(* CODESYS project plc_chalet_base.library
   Title: CHALET_BaseComponents
   Version: 3.2.4
   Placeholder: CHALET_BaseComponents
   Company: Beckhoff CH

Project tree, tasks and I/O mapping:
  libraries: Tc2_EtherCAT, * (Beckhoff Automation GmbH); Tc2_Standard, 3.3.3.0 (Beckhoff Automation GmbH); Tc2_System, 3.4.25.0 (Beckhoff Automation GmbH); Tc2_Utilities, 3.3.52.0 (Beckhoff Automation GmbH); Tc3_EventLogger, 3.1.30.0 (Beckhoff Automation GmbH); Tc3_Module, 3.3.21.0 (Beckhoff Automation GmbH)
  COMPONENTs/
    CoE-Access/
      internal/
        function block FB_CoE_Base [ST]: cbBufLen, Index, pSrcBuf, SubIndex, Error, FB_init, ReadDone, Update, WriteDone
        interface I_AdsAddr: NetId, Port
      function block FB_CoE_BOOL [ST]: cbBufLen, pSrcBuf, Value
      function block FB_CoE_BYTE [ST]: cbBufLen, pSrcBuf, Value
      function block FB_CoE_Connection [ST]: Mapped, NetId, Port
      function block FB_CoE_UDINT [ST]: cbBufLen, pSrcBuf, Value
      function block FB_CoE_UINT [ST]: cbBufLen, pSrcBuf, Value
    Feedback/
      function block FB_CH_Feedback [ST]: ActiveCommand, Busy, Done, Error, ErrorId, HR, LastCommandAccepted
      interface I_CH_Feedback: ActiveCommand, Busy, Done, Error, ErrorId, HR, LastCommandAccepted
    HR/
      function CheckNotOk [ST]
      function CheckOk [ST]
      function GetMostSignificant [ST]
    List/
      CD_CH_List
      function block FB_CH_List [ST]: FindLUID, FindOID, FindOIDString, ResetIterator, RestoreIterator, AddList, Clear, Duplicate, Initialize, IsEmpty, IsFull, Size, Update, AddObject, FindObject, GetNextObject, GetRandomObject, HasNextObject, RemoveObject
      interface I_CH_LIST: FindLUID, FindOID, FindOIDString, GetNextObject, GetRandomObject, HasNextObject, IsEmpty, IsFull, ResetIterator, RestoreIterator, Size
    Object/
      CD_CH_Object
      function block FB_CH_Object [ST]: FB_init, Initialize, LUID, OID, TaskIndex, Update
      interface I_CH_Object: Initialize, LUID, OID, Update
    global variables GVL_Datatypes
  global variables BaseParameterlist
  00000000-0000-0000-0000-000000000000|LICENSE.md
  LICENSE.md
*)

// COMPONENTs/GVL_Datatypes
{attribute 'qualified_only'}
VAR_GLOBAL CONSTANT
	// SINT
	cMaxSint	: SINT 		:= 127; // Largest SINT number
    cMinSint	: SINT 		:= -128; // Smallest SINT number

	// USINT
	cMaxUsint	: USINT 	:= 255; // Largest USINT number
    cMinUSint	: USINT 	:= 0; // Smallest USINT number

	// INT
	cMaxInt		: INT 		:= 32_767; // Largest INT number
    cMinInt		: INT 		:= -32_768; // Smallest INT number

	// UINT
	cMaxUint	: UINT 		:= 65_535; // Largest UINT number
    cMinUnit	: UINT 		:= 0; // Smallest UINT number

	// DINT
	cMaxDint	: DINT 		:= 2_147_483_647; // Largest DINT number
    cMinDint	: DINT 		:= -2_147_483_648; // Smallest DINT number

	// UDINT
	cMaxUdint	: UDINT 	:= 4_294_967_295; // Largest UDINT number
    cMinUdint	: UDINT		:= 0; // Smallest UDINT number

	// LINT
	cMaxLint	: LINT 		:= 9_223_372_036_854_775_807; // Largest LINT number
    cMinBLint	: LINT 		:= -9_223_372_036_854_775_808; // Smallest LINT number

	// ULINT
	cMaxUlint	: ULINT 	:= 18_446_744_073_709_551_615; // Largest ULINT number
    cMinUlint	: ULINT 	:= 0; // Smallest ULINT number

	// BYTE
	cMaxByte	: BYTE 		:= 255; // Largest BYTE number
    cMinByte	: BYTE 		:= 0; // Smallest BYTE number

	// WORD
	cMaxWord	: WORD 		:= 65_535; // Largest WORD number
    cMinWord	: WORD 		:= 0; // Smallest WORD number

	// DWORD
	cMaxDword	: DWORD 	:= 4_294_967_295; // Largest DWORD number
    cMinDword	: DWORD 	:= 0; // Smallest DWORD number

	// LWORD
	cMaxLword	: LWORD 	:= 18_446_744_073_709_551_615; // Largest LWORD number
    cMinLword	: LWORD 	:= 0; // Smallest LWORD number
	
	// REAL
	cMaxReal	: REAL 		:= 3.402823E+38; // Largest REAL number
    cMinReal	: REAL 		:= -3.402823E+38; // Smallest REAL number
	
	// LREAL
    cMaxLreal	: LREAL 	:= 1.7976931348623157E+308; // Largest LREAL number
    cMinLreal	: LREAL 	:= -1.7976931348623157E+308; // Smallest LREAL number
	
    // DATE
    cMaxDate   	: DATE    	:= DATE#2106-2-7; // Maximum DATA
    cMinDate   	: DATE     	:= DATE#1970-1-1; // Minimum DATE
	
	// TIME
	cMaxTime	: TIME  	:= T#49D17H2M47S295MS; // Longest TIME duration
	cMinTime 	: TIME  	:= TO_TIME(0);	// Shortest TIME duration
	
	// LTIME
	cMaxLtime	: LTIME 	:= LTIME#213503D23H34M33S709MS551US615NS; // Longest LTIME duration
	cMinLtime 	: LTIME  	:= TO_LTIME(0); // Shortest LTIME duration
	
    // Date and time
    cMaxDataAndTime  : DATE_AND_TIME  := DATE_AND_TIME#2106-02-07-06:28:15; // Maximum DATA_AND_DATE
    cMinDataAndTime  : DATE_AND_TIME  := DATE_AND_TIME#1970-1-1-0:0:0; // Minimum DATA_AND_DATE

    // Time of day
    cMaxTimeOfDay 	: TIME_OF_DAY    := TIME_OF_DAY#23:59:59.999; // Largest TIME_OF_DAY
    cMinTimeOfDay 	: TIME_OF_DAY    := TIME_OF_DAY#0:0:0; // Smallest TIME_OF_DAY

END_VAR

// BaseParameterlist
{attribute 'qualified_only'}
VAR_GLOBAL CONSTANT
	(*Maximum length of List*)
	MAX_OBJECTS 			: UDINT := 150;
	
	(*Maximum CoE-Read at same time*)
	MAX_COE_READ 			: UDINT := 20;
	
	(*Maximum CoE-Write at same time*)
	MAX_COE_WRITE 			: UDINT := 20;
	
	
END_VAR

// COMPONENTs/CoE-Access/internal/FB_CoE_Base
(* This FB is abstract and is the base class  *)
FUNCTION_BLOCK ABSTRACT FB_CoE_Base EXTENDS FB_CH_Object
VAR
	//Coe Connector
	{attribute 'hide'}
	ipCoeConnection	: I_AdsAddr;
	{attribute 'hide'}
	bErrorInvalideInterface : BOOL;
	
	//Parameter index
	{attribute 'hide'}
    nIndex     : WORD; (* CoE Object Index *)
	{attribute 'hide'}
    nSubIndex  : BYTE; (* Subindex of CoE Object *)

	//Read/write 
	{attribute 'hide'}
	bReadDone : BOOL;
	{attribute 'hide'}
	fbCoeRead : FB_EcCoeSdoRead;
	{attribute 'hide'}
	nSeqRead : UINT;
	{attribute 'hide'}
	bReadError : BOOL;
	
	{attribute 'hide'}
	bWriteDone : BOOL := TRUE;
	{attribute 'hide'}
	fbCoeWrite : FB_EcCoeSdoWrite;
	{attribute 'hide'}
	nSeqWrite : UINT;
	{attribute 'hide'}
	bWriteError : BOOL;
	
	{attribute 'hide'}
	fbDelayOnError : TON := ( PT:= T#10S);
END_VAR
VAR_STAT
	nCtsCoeObject : UDINT;
	nCtsReadActive : UDINT;
	nCtsWriteActive : UDINT;
END_VAR

PROPERTY PROTECTED ABSTRACT cbBufLen : UDINT
GET
END_GET
END_PROPERTY

PROPERTY PRIVATE Index : WORD
GET
END_GET
END_PROPERTY

PROPERTY PROTECTED ABSTRACT pSrcBuf : PVOID
GET
END_GET
END_PROPERTY

PROPERTY PRIVATE SubIndex : BYTE
GET
END_GET
END_PROPERTY

{attribute 'monitoring':='call'}
PROPERTY Error : BOOL
GET
Error := THIS^.bReadError OR THIS^.bWriteError OR THIS^.bErrorInvalideInterface;
END_GET
END_PROPERTY

METHOD FB_init : BOOL
VAR_INPUT
	bInitRetains : BOOL; // if TRUE, the retain variables are initialized (warm start / cold start)
	bInCopyCode : BOOL;  // if TRUE, the instance afterwards gets moved into the copy code (online change)
	
	ipCoeConnection	: I_AdsAddr;
    nIndex     : WORD; 	(* CoE Object Index *)
    nSubIndex  : BYTE; 		(* Subindex of CoE Object *)
END_VAR

VAR_INST
	{attribute 'hide'}
	bFBInitCalledOnce : BOOL; //Do the following code once during start up and not during onlinechange
END_VAR
//Do the following code once during start up and not during onlinechange
IF NOT bFBInitCalledOnce THEN 
	nCtsCoeObject := nCtsCoeObject +1;
	
	THIS^.ipCoeConnection := ipCoeConnection;
	THIS^.nIndex 		:= nIndex;
	THIS^.nSubIndex 	:= nSubIndex;
END_IF

bFBInitCalledOnce := TRUE;
END_METHOD

{attribute 'monitoring':='call'}
PROPERTY ReadDone : BOOL
GET
ReadDone := bReadDone;
END_GET
SET
//Only allow set to FALSE
IF NOT ReadDone THEN
	bReadDone := FALSE;
END_IF
END_SET
END_PROPERTY

METHOD Update : HRESULT
IF ipCoeConnection = 0 THEN
	bErrorInvalideInterface := TRUE;
	RETURN;
END_IF


(*--- Read ---*)
CASE nSeqRead OF
	0: //Start/Restart if required
		IF NOT bReadDone  AND bWriteDone(* Write has higher priority*) AND (nCtsReadActive < BaseParameterlist.MAX_COE_READ) AND (nSeqWrite = 0) THEN
			fbCoeRead.bExecute := TRUE; // Rising edge	
			nCtsReadActive := nCtsReadActive +1;	
			nSeqRead := 1;
		END_IF
	
	1: //Check if done or error
		IF fbCoeRead.bError THEN
			//Error
			nSeqRead := 99;
			bReadError := TRUE;
			fbDelayOnError.IN := TRUE;
			nCtsReadActive := nCtsReadActive -1;	
			
		ELSIF NOT fbCoeRead.bBusy AND NOT fbCoeRead.bError THEN
			//Done
			THIS^.bReadDone := TRUE;
			nSeqRead := 0;
			bReadError := FALSE;
			nCtsReadActive := nCtsReadActive -1;	
		END_IF	
		
	99: // Delay on error to reduce amount of errors
		IF fbDelayOnError.Q THEN
			fbDelayOnError.IN := FALSE;
			nSeqRead := 0;
		END_IF
END_CASE

IF NOT THIS^.bReadDone THEN
	fbCoeRead(
		sNetId		:= ipCoeConnection.NetId,
		nSlaveAddr	:= ipCoeConnection.port,
		nSubIndex	:= THIS^.nSubIndex, 
		nIndex		:= THIS^.nIndex, 
		pDstBuf		:= THIS^.pSrcBuf, 
		cbBufLen	:= THIS^.cbBufLen);
		
	//Prepare for next rising edge
	fbCoeRead.bExecute := FALSE;
END_IF



(*--- Write ---*)
CASE nSeqWrite OF
	0: //Start/Restart if required
		IF NOT bWriteDone AND (nCtsWriteActive < BaseParameterlist.MAX_COE_WRITE) AND (nSeqRead = 0) THEN
			fbCoeWrite.bExecute := TRUE; // Rising edge	
			nCtsWriteActive := nCtsWriteActive +1;	
			nSeqWrite := 1;
		END_IF
	
	1: //Check if done or error
		IF fbCoeWrite.bError THEN
			//Error
			nSeqWrite := 99;
			bWriteError := TRUE;
			fbDelayOnError.IN := TRUE;
			nCtsWriteActive := nCtsWriteActive -1;	
			
		ELSIF NOT fbCoeWrite.bBusy AND NOT fbCoeWrite.bError THEN
			//Done
			THIS^.bWriteDone := TRUE;
			nSeqWrite := 0;
			bWriteError := FALSE;
			nCtsWriteActive := nCtsWriteActive -1;	
		END_IF	
		
	99: // Delay on error to reduce amount of errors
		IF fbDelayOnError.Q THEN
			fbDelayOnError.IN := FALSE;
			nSeqWrite := 0;
		END_IF		

END_CASE

IF NOT bWriteDone THEN
	fbCoeWrite(
		sNetId		:= ipCoeConnection.netId, 
		nSlaveAddr	:= ipCoeConnection.port,
		nSubIndex	:= THIS^.nSubIndex, 
		nIndex		:= THIS^.nIndex, 
		pSrcBuf		:= THIS^.pSrcBuf, 
		cbBufLen	:= THIS^.cbBufLen);		
		
	//Prepare for next rising edge
	fbCoeWrite.bExecute := FALSE;
END_IF

//Update
fbDelayOnError();
END_METHOD

{attribute 'monitoring':='call'}
PROPERTY WriteDone : BOOL
GET
WriteDone := bWriteDone;
END_GET
SET
//Only allow set to FALSE
IF NOT WriteDone THEN
	bWriteDone := FALSE;
END_IF
END_SET
END_PROPERTY

END_FUNCTION_BLOCK

// COMPONENTs/Object/FB_CH_Object
FUNCTION_BLOCK FB_CH_Object IMPLEMENTS I_CH_Object
VAR
	fbSourceInfo : FB_TcSourceInfo;
	
	{attribute 'hide'}
	nTaskIndex : BYTE; //Used in TwinCAT_SystemInfoVarList._TaskInfo
END_VAR

METHOD FB_init : BOOL
VAR_INPUT
	bInitRetains : BOOL; // if TRUE, the retain variables are initialized (warm start / cold start)
	bInCopyCode : BOOL;  // if TRUE, the instance afterwards gets moved into the copy code (online change)
END_VAR
VAR
	fbGetCurTaskIdx  : GETCURTASKINDEX;
END_VAR
fbGetCurTaskIdx();
THIS^.nTaskIndex := fbGetCurTaskIdx.Index;
END_METHOD

METHOD Initialize : HRESULT
Initialize := S_OK;
END_METHOD

{attribute 'monitoring':='call'}
PROPERTY LUID : STRING //Locally unique identifier
GET
LUID := THIS^.fbSourceInfo.sName;
END_GET
END_PROPERTY

{attribute 'monitoring':='call'}
PROPERTY OID : OTCID //Object ID
GET
OID := 0;
END_GET
END_PROPERTY

PROPERTY PROTECTED TaskIndex : BYTE //Used in TwinCAT_SystemInfoVarList._TaskInfo
GET
TaskIndex := THIS^.nTaskIndex;
END_GET
END_PROPERTY

METHOD Update : HRESULT
VAR_INPUT
END_VAR
Update := S_OK;
END_METHOD

END_FUNCTION_BLOCK

// COMPONENTs/Object/I_CH_Object
INTERFACE I_CH_Object EXTENDS __SYSTEM.IQueryInterface

METHOD Initialize : HRESULT
END_METHOD

{attribute 'monitoring':='call'}
PROPERTY LUID : STRING //Locally unique identifier
GET
END_GET
END_PROPERTY

{attribute 'monitoring':='call'}
PROPERTY OID : OTCID //Object ID
GET
END_GET
END_PROPERTY

METHOD Update : HRESULT
VAR_INPUT
END_VAR
END_METHOD

END_INTERFACE

// COMPONENTs/CoE-Access/internal/I_AdsAddr
INTERFACE I_AdsAddr

{attribute 'monitoring':='call'}
PROPERTY NetId : T_AmsNetID
GET
END_GET
END_PROPERTY

{attribute 'monitoring':='call'}
PROPERTY Port : WORD
GET
END_GET
END_PROPERTY

END_INTERFACE

// COMPONENTs/CoE-Access/FB_CoE_BOOL
{attribute 'no_explicit_call' := 'Do not call the body - Stick to OOP'}
FUNCTION_BLOCK FB_CoE_BOOL EXTENDS FB_CoE_Base
VAR
	{attribute 'hide'}
	nValue : BOOL;
END_VAR

PROPERTY PROTECTED cbBufLen : UDINT
GET
cbBufLen := SIZEOF(nValue);
END_GET
END_PROPERTY

PROPERTY PROTECTED pSrcBuf : PVOID
GET
pSrcBuf := ADR(nValue);
END_GET
END_PROPERTY

{attribute 'monitoring':='call'}
PROPERTY Value : BOOL
GET
Value := nValue;
END_GET
SET
nValue := Value;

//Trigger a new write cycle
THIS^.bWriteDone 	:= FALSE;
END_SET
END_PROPERTY

END_FUNCTION_BLOCK

// COMPONENTs/CoE-Access/FB_CoE_BYTE
{attribute 'no_explicit_call' := 'Do not call the body - Stick to OOP'}
FUNCTION_BLOCK FB_CoE_BYTE EXTENDS FB_CoE_Base
(* 
   FB_init:
	(	ipCoeConnection := fbCoeConnection, (*each EC-Slave needs one FB_CoE_Connection*)
		nIndex     		:= 16#8010, (* CoE Object Index *)
		nSubIndex  		:= 16#11 (* Subindex of CoE Object *));
 *)
VAR
	{attribute 'hide'}
	nValue : BYTE;
END_VAR

PROPERTY PROTECTED cbBufLen : UDINT
GET
cbBufLen := SIZEOF(nValue);
END_GET
END_PROPERTY

PROPERTY PROTECTED pSrcBuf : PVOID
GET
pSrcBuf := ADR(nValue);
END_GET
END_PROPERTY

{attribute 'monitoring':='call'}
PROPERTY Value : BYTE
GET
Value := nValue;
END_GET
SET
nValue := Value;

//Trigger a new write cycle
THIS^.bWriteDone 	:= FALSE;
END_SET
END_PROPERTY

END_FUNCTION_BLOCK

// COMPONENTs/CoE-Access/FB_CoE_Connection
(* This FB must be instantiated once per EtherCat slave. 
It is used to generate the PLC process image required to read the ADS address + port from the terminal. 
This information is then transferred to the individual FBs for the registers *)
{attribute 'no_explicit_call' := 'Do not call the body - Stick to OOP'}
FUNCTION_BLOCK  FB_CoE_Connection IMPLEMENTS I_AdsAddr
VAR
	AdsAddr AT %I* : AMSADDR;
END_VAR

{attribute 'monitoring':='call'}
PROPERTY Mapped : BOOL
GET
VAR
	bNotMapped : BOOL;
END_VAR
bNotMapped := F_GetMappingStatus(ADR(THIS^.AdsAddr), SIZEOF(THIS^.AdsAddr)) <> EPlcMappingStatus.MS_Mapped;

Mapped := NOT bNotMapped;
END_GET
END_PROPERTY

{attribute 'monitoring':='call'}
PROPERTY NetId : T_AmsNetID
GET
//Convert number to string
NetId := F_CreateAmsNetId( AdsAddr.netId );
END_GET
END_PROPERTY

{attribute 'monitoring':='call'}
PROPERTY Port : WORD
GET
Port := AdsAddr.port;
END_GET
END_PROPERTY

END_FUNCTION_BLOCK

// COMPONENTs/CoE-Access/FB_CoE_UDINT
{attribute 'no_explicit_call' := 'Do not call the body - Stick to OOP'}
FUNCTION_BLOCK FB_CoE_UDINT EXTENDS FB_CoE_Base
(* 
   FB_init:
	(	ipCoeConnection := fbCoeConnection, (*each EC-Slave needs one FB_CoE_Connection*)
		nIndex     		:= 16#8010, (* CoE Object Index *)
		nSubIndex  		:= 16#11 (* Subindex of CoE Object *));
 *)
VAR
	{attribute 'hide'}
	nValue : UDINT;
END_VAR

PROPERTY PROTECTED cbBufLen : UDINT
GET
cbBufLen := SIZEOF(nValue);
END_GET
END_PROPERTY

PROPERTY PROTECTED pSrcBuf : PVOID
GET
pSrcBuf := ADR(nValue);
END_GET
END_PROPERTY

{attribute 'monitoring':='call'}
PROPERTY Value : UDINT
GET
Value := nValue;
END_GET
SET
nValue := Value;

//Trigger a new write cycle
THIS^.bWriteDone 	:= FALSE;
END_SET
END_PROPERTY

END_FUNCTION_BLOCK

// COMPONENTs/CoE-Access/FB_CoE_UINT
{attribute 'no_explicit_call' := 'Do not call the body - Stick to OOP'}
FUNCTION_BLOCK FB_CoE_UINT EXTENDS FB_CoE_Base
(* 
   FB_init:
	(	ipCoeConnection := fbCoeConnection, (*each EC-Slave needs one FB_CoE_Connection*)
		nIndex     		:= 16#8010, (* CoE Object Index *)
		nSubIndex  		:= 16#11 (* Subindex of CoE Object *));
 *)
VAR
	{attribute 'hide'}
	nValue : UINT;
END_VAR

PROPERTY PROTECTED cbBufLen : UDINT
GET
cbBufLen := SIZEOF(nValue);
END_GET
END_PROPERTY

PROPERTY PROTECTED pSrcBuf : PVOID
GET
pSrcBuf := ADR(nValue);
END_GET
END_PROPERTY

{attribute 'monitoring':='call'}
PROPERTY Value : UINT
GET
Value := nValue;
END_GET
SET
nValue := Value;

//Trigger a new write cycle
THIS^.bWriteDone 	:= FALSE;
END_SET
END_PROPERTY

END_FUNCTION_BLOCK

// COMPONENTs/Feedback/FB_CH_Feedback
FUNCTION_BLOCK FB_CH_Feedback IMPLEMENTS I_CH_Feedback
VAR
    {attribute 'hide'}
    _hr : HRESULT;
    {attribute 'hide'}
    _activeCommand : STRING;
    {attribute 'hide'}
    _lastCommandAccepted : BOOL;
END_VAR

{attribute 'monitoring' := 'call'}
PROPERTY ActiveCommand : STRING;
GET
ActiveCommand := THIS^._ActiveCommand;
END_GET
SET
THIS^._ActiveCommand 		:= ActiveCommand;
END_SET
END_PROPERTY

{attribute 'monitoring' := 'call'}
(* Indicates a busy command, i.e. command is being processed, waiting for execution, or already executing (= also active). *)
PROPERTY Busy : BOOL
GET
Busy := (THIS^._hr = S_PENDING);
END_GET
SET
IF Busy THEN
	THIS^._hr := S_PENDING;
END_IF
END_SET
END_PROPERTY

{attribute 'monitoring' := 'call'}
(* Indicates the command is done, i.e. execution of the command finished successfully. *)
PROPERTY Done : BOOL
GET
Done := NOT THIS^.Busy AND NOT THIS^.Error;
END_GET
SET
IF Done THEN
	THIS^._hr := S_OK;
END_IF
END_SET
END_PROPERTY

{attribute 'monitoring' := 'call'}
(* Indicates the command has an error. *)
PROPERTY Error : BOOL
GET
Error := FAILED(THIS^._hr);
END_GET
END_PROPERTY

{attribute 'monitoring' := 'call'}
(* Indicates the error id of the command error. *)
PROPERTY ErrorId : UDINT
GET
ErrorId := DWORD_TO_UDINT(DINT_TO_DWORD(THIS^._hr) AND 16#0000FFFF); //only return the last two byte with the error Id

//515 means busy and is not an Error
IF ErrorId = 515 THEN
	ErrorId := 0;
END_IF
END_GET
SET
VAR
	//A failed execution is indicated by a NEGATIVE code, or in hexadecimal notation the first digit is >= 8.
	nErrorCodeSign : UDINT := 16#80000000;
END_VAR
IF ErrorId <> 0 THEN
	THIS^._hr := TO_DINT(nErrorCodeSign + ErrorId);
END_IF
END_SET
END_PROPERTY

{attribute 'monitoring' := 'call'}
PROPERTY HR : HRESULT
GET
HR := THIS^._hr;
END_GET
SET
THIS^._hr := HR;
END_SET
END_PROPERTY

{attribute 'monitoring' := 'call'}
PROPERTY LastCommandAccepted : BOOL
GET
LastCommandAccepted := THIS^._lastCommandAccepted;
END_GET
SET
THIS^._lastCommandAccepted := LastCommandAccepted;
END_SET
END_PROPERTY

END_FUNCTION_BLOCK

// COMPONENTs/Feedback/I_CH_Feedback
INTERFACE I_CH_Feedback

{attribute 'monitoring' := 'call'}
PROPERTY ActiveCommand : STRING;
GET
END_GET
END_PROPERTY

{attribute 'monitoring' := 'call'}
(* Indicates a busy command, i.e. command is being processed, waiting for execution, or already executing (= also active). *)
PROPERTY Busy : BOOL
GET
END_GET
END_PROPERTY

{attribute 'monitoring' := 'call'}
(* Indicates the command is done, i.e. execution of the command finished successfully. *)
PROPERTY Done : BOOL
GET
END_GET
END_PROPERTY

{attribute 'monitoring' := 'call'}
(* Indicates the command has an error. *)
PROPERTY Error : BOOL
GET
END_GET
END_PROPERTY

{attribute 'monitoring' := 'call'}
(* Indicates the error id of the command error. *)
PROPERTY ErrorId : UDINT
GET
END_GET
END_PROPERTY

{attribute 'monitoring' := 'call'}
PROPERTY HR : HRESULT
GET
END_GET
END_PROPERTY

{attribute 'monitoring' := 'call'}
PROPERTY LastCommandAccepted : BOOL
GET
END_GET
END_PROPERTY

END_INTERFACE

// COMPONENTs/HR/CheckNotOk
FUNCTION CheckNotOk : BOOL
VAR_INPUT
	hr : HRESULT;
END_VAR

CheckNotOk := (hr <> S_OK);

END_FUNCTION

// COMPONENTs/HR/CheckOk
FUNCTION CheckOk : BOOL
VAR_INPUT
	hr : HRESULT;
END_VAR

CheckOk := (hr = S_OK);

END_FUNCTION

// COMPONENTs/HR/GetMostSignificant
(*
	Return the most significant HRESULT input (hr1 or hr2).
	Example: if hr1:= S_Pending and hr2 := S_OK, then return S_Pending 
	Priority:(Error(incl. code) > Error(empty code) > S_WATCHDOGTIMEOUT > S_PENDING > S_FALSE > S_OK)
*)
FUNCTION GetMostSignificant : HRESULT
VAR_INPUT
	hr1 : HRESULT; //top priority if both hr1 and hr2 have an error code return this
	hr2 : HRESULT; //second priority if both hr1 and hr2 have an error code return hr1
END_VAR

//hr1 has an Error(incl. errorcode) 
IF hr1.31 AND ((TO_DWORD(hr1) AND 16#FFF) > 0) THEN
	GetMostSignificant := hr1;

//hr2 has an Error(incl. errorcode) 
ELSIF hr2.31 AND ((TO_DWORD(hr2) AND 16#FFF) > 0) THEN
	GetMostSignificant := hr2;

//hr1 has an Error(empty errorcode)
ELSIF hr1.31 THEN
	GetMostSignificant := hr1;

//hr2 has an Error(empty errorcode)
ELSIF hr2.31 THEN
	GetMostSignificant := hr2;
	
//hr1 has a higher SUCCESS code than hr2. (S_WATCHDOGTIMEOUT > S_PENDING > S_FALSE > S_OK)
ELSIF hr1 >= hr2 THEN
	GetMostSignificant := hr1;

//hr2 has a higher SUCCESS code than hr1. (S_WATCHDOGTIMEOUT > S_PENDING > S_FALSE > S_OK)
ELSE 
	GetMostSignificant := hr2;	
	
END_IF

END_FUNCTION

// COMPONENTs/List/FB_CH_List
FUNCTION_BLOCK FB_CH_List EXTENDS FB_CH_Object IMPLEMENTS I_CH_LIST
VAR
	{attribute 'hide'}
	nObjectCount			: UDINT;
	{attribute 'hide'}
	nIdxNextObject			: UDINT;
	{attribute 'hide'}
	nIdxLastRestoreValues : ARRAY [0..(MAX_CTS_RESTORE_VALUES+1)] OF UDINT;
	{attribute 'hide'}
	nIdxRestore				: UDINT;
	aObjects				: ARRAY [1..BaseParameterlist.MAX_OBJECTS] OF I_CH_Object;
END_VAR
VAR CONSTANT
	{attribute 'hide'}
	MAX_CTS_RESTORE_VALUES : UINT := 9;
END_VAR

METHOD PUBLIC FindLUID : I_CH_OBJECT
VAR_INPUT
	sLUID	: STRING;
END_VAR
VAR
	nIdx : UDINT;
END_VAR
FOR nIdx := 1 TO nObjectCount DO
	IF aObjects[nIdx] <> 0 AND_THEN aObjects[nIdx].LUID = sLUID THEN
		FindLUID := aObjects[nIdx];
		EXIT;
	END_IF
END_FOR
END_METHOD

METHOD FindOID : I_CH_OBJECT
VAR_INPUT
	oOID	: OTCID;
END_VAR
VAR
	nIdx : UDINT;
END_VAR
FOR nIdx := 1 TO nObjectCount DO
	IF aObjects[nIdx] <> 0 AND_THEN aObjects[nIdx].OID = oOID THEN
		FindOID := aObjects[nIdx];
		EXIT;
	END_IF
END_FOR
END_METHOD

METHOD FindOIDString : I_CH_OBJECT
VAR_INPUT
	sOID	: STRING;
END_VAR
VAR
	nIdx : UDINT;
END_VAR
FOR nIdx := 1 TO nObjectCount DO
	IF aObjects[nIdx] <> 0 AND_THEN DWORD_TO_HEXSTR(TO_DWORD(aObjects[nIdx].OID),0,FALSE) = sOID THEN
		FindOIDString := aObjects[nIdx];
		EXIT;
	END_IF
END_FOR
END_METHOD

METHOD PUBLIC ResetIterator : BOOL
VAR_INPUT
END_VAR
//Store the last few index for later restore if required - Shift array +1 step
MEMMOVE(srcAddr 	:= ADR(nIdxLastRestoreValues[0]), 
		destAddr 	:= ADR(nIdxLastRestoreValues[1]), 
		n 			:= (SIZEOF(nIdxNextObject)*MAX_CTS_RESTORE_VALUES));

//Store the last few index for later restore if required - Store last value
nIdxLastRestoreValues[0] := nIdxNextObject;


nIdxNextObject := 0;
END_METHOD

//Restore the iterator to the value before the last reset. This is necessary if several white loops are placed inside each other
METHOD PUBLIC RestoreIterator : BOOL
VAR_INPUT
END_VAR
//Store the last few index for later restore if required - Restore
nIdxNextObject := nIdxLastRestoreValues[0];

//Store the last few index for later restore if required - Shift array -1 step
MEMMOVE(srcAddr 	:= ADR(nIdxLastRestoreValues[1]), 
		destAddr 	:= ADR(nIdxLastRestoreValues[0]), 
		n 			:= (SIZEOF(nIdxNextObject)*MAX_CTS_RESTORE_VALUES));
END_METHOD

//Add all objects from the list in to this list
METHOD PUBLIC AddList : HRESULT
VAR_INPUT
	ipList	: I_CH_List;
END_VAR
VAR
	hr : HRESULT;
END_VAR
IF ipList = 0 THEN
	AddList := S_FALSE;
	RETURN;
END_IF

ipList.ResetIterator();
WHILE ipList.HasNextObject() DO
	hr := THIS^.AddObject(ipList.GetNextObject());
	IF hr <> S_OK THEN
		//Error
		AddList := hr;
		RETURN;
	END_IF
END_WHILE
ipList.RestoreIterator();
END_METHOD

METHOD PUBLIC Clear : BOOL
VAR
	nIdx : UDINT;
END_VAR
FOR nIdx := 1 TO BaseParameterlist.MAX_OBJECTS DO
	aObjects[nIdx] := NULL;
END_FOR

nObjectCount	:= 0;
nIdxNextObject	:= 0;
END_METHOD

METHOD Duplicate : BOOL
VAR_INPUT
	ipListCopyFrom : I_CH_LIST;
END_VAR
VAR
	ipThisList : I_CH_LIST := THIS^;
END_VAR
//New list equals this list
IF ipListCopyFrom = ipThisList THEN
	//Do Nothing - Successfull
	Duplicate := TRUE;
	RETURN;
END_IF


THIS^.Clear();

// Invalide input
IF ipListCopyFrom = 0 THEN
	Duplicate := FALSE;
	RETURN;
END_IF


// This list is to small
IF ipListCopyFrom.Size > BaseParameterlist.MAX_OBJECTS THEN
	Duplicate := FALSE;
	RETURN;
END_IF



ipListCopyFrom.ResetIterator();
WHILE ipListCopyFrom.HasNextObject() DO
	THIS^.AddObject(ipListCopyFrom.GetNextObject());
END_WHILE
ipListCopyFrom.RestoreIterator();


Duplicate := TRUE;
END_METHOD

METHOD Initialize : HRESULT //This method calls the respective Initialize method of all contained objects
VAR_INPUT
END_VAR
VAR
	hr : HRESULT;
	nIdx : UDINT;
END_VAR
//FOR each element
FOR nIdx := 1 TO nObjectCount DO
	// DO Init
	hr := GetMostSignificant(hr, aObjects[nIdx].Initialize());
END_FOR


Initialize := hr;
END_METHOD

{attribute 'monitoring':='call'}
PROPERTY PUBLIC IsEmpty : BOOL
GET
IsEmpty := (nObjectCount = 0);
END_GET
END_PROPERTY

{attribute 'monitoring':='call'}
PROPERTY PUBLIC IsFull : BOOL
GET
IsFull := (nObjectCount = BaseParameterlist.MAX_OBJECTS);
END_GET
END_PROPERTY

{attribute 'monitoring':='call'}
PROPERTY PUBLIC Size : UDINT
GET
Size := nObjectCount;
END_GET
END_PROPERTY

METHOD Update : HRESULT //This method calls the respective update method of all contained objects
VAR
	hr : HRESULT;
	nIdx : UDINT;
END_VAR
//FOR each element
FOR nIdx := 1 TO nObjectCount DO
	// DO Update
	hr := GetMostSignificant(hr, aObjects[nIdx].Update());
END_FOR

Update := hr;
END_METHOD

METHOD PUBLIC AddObject : HRESULT
VAR_INPUT
	iChObject	: I_CH_Object;
END_VAR
VAR_INST
	{attribute 'hide'}
	fbAlarmListFull : FB_TcAlarm;
END_VAR
IF nObjectCount >= BaseParameterlist.MAX_OBJECTS THEN
	fbAlarmListFull.CreateEx(stEventEntry:= TC_EVENTS.CHALET_Base_Events.ListIsFull, 
							ipSourceInfo := THIS^.fbSourceInfo, 
							bWithConfirmation := FALSE);
	fbAlarmListFull.Raise(0);
	AddObject := S_FALSE;
	RETURN;
END_IF

IF iChObject = 0 THEN
	AddObject := S_FALSE;
	RETURN;
END_IF

nObjectCount := nObjectCount + 1;
aObjects[nObjectCount] := iChObject;

AddObject := S_OK;
END_METHOD

METHOD PUBLIC FindObject : BOOL
VAR_INPUT
	iChObject	: I_CH_Object;
END_VAR
VAR
	nIdx : UDINT;
END_VAR
//Check array until a match
FOR nIdx := 1 TO THIS^.nObjectCount DO
	IF THIS^.aObjects[nIdx] = iChObject THEN
		FindObject := TRUE;
		EXIT;
	END_IF
END_FOR
END_METHOD

METHOD PUBLIC GetNextObject : I_CH_Object
VAR_INPUT
END_VAR
nIdxNextObject := nIdxNextObject + 1;


IF nIdxNextObject > nObjectCount THEN
	//Error!
	//Todo: Errormessage
	GetNextObject := 0;
	RETURN;
END_IF




GetNextObject := aObjects[nIdxNextObject];
END_METHOD

METHOD GetRandomObject : I_CH_Object
VAR_INPUT
END_VAR

VAR_INST
	{attribute 'hide'}
	fbDRAN : DRAND;
END_VAR

VAR
	nRandomIdx : UDINT;
END_VAR
//Check if not Empty
IF UDINT_TO_BOOL(nObjectCount) THEN
	// Generate number 0..1
	fbDRAN(Seed:= 42);
	
	// 1..Size   = ((0..1)*(Size-1))+1
	nRandomIdx := LREAL_TO_UDINT(fbDRAN.Num * (nObjectCount-1))+1;
	
	GetRandomObject := aObjects[nRandomIdx];
	
END_IF
END_METHOD

METHOD PUBLIC HasNextObject : BOOL
VAR_INPUT
END_VAR
HasNextObject := (nIdxNextObject < nObjectCount);
END_METHOD

METHOD PUBLIC RemoveObject : BOOL
VAR_INPUT
	iChObject	: I_CH_Object;
END_VAR

VAR
	nIdx			: UDINT;
END_VAR
RemoveObject := FALSE;

IF iChObject = 0 THEN
	RETURN;
END_IF

IF NOT THIS^.FindObject(iChObject) THEN
	RETURN;
END_IF

FOR nIdx := 1 TO nObjectCount DO
	IF aObjects[nIdx] = iChObject THEN
		aObjects[nIdx] := NULL;	
		
		nObjectCount := nObjectCount - 1;
		
		// Fill up the empty slot
		MEMMOVE(ADR(aObjects[nIdx]), ADR(aObjects[nIdx + 1]), SIZEOF(aObjects[nIdx]) * (BaseParameterlist.MAX_OBJECTS - nIdx));
	
		RemoveObject := TRUE;
		EXIT;
	END_IF
END_FOR
END_METHOD

END_FUNCTION_BLOCK

// COMPONENTs/List/I_CH_LIST
INTERFACE I_CH_LIST

METHOD PUBLIC FindLUID : I_CH_OBJECT
VAR_INPUT
	sLUID	: STRING;
END_VAR
END_METHOD

METHOD FindOID : I_CH_OBJECT
VAR_INPUT
	oOID	: OTCID;
END_VAR
END_METHOD

METHOD FindOIDString : I_CH_OBJECT
VAR_INPUT
	sOID	: STRING;
END_VAR
END_METHOD

METHOD PUBLIC GetNextObject : I_CH_Object
VAR_INPUT
END_VAR
END_METHOD

METHOD GetRandomObject : I_CH_Object
VAR_INPUT
END_VAR
END_METHOD

METHOD PUBLIC HasNextObject : BOOL
VAR_INPUT
END_VAR
END_METHOD

{attribute 'monitoring':='call'}
PROPERTY PUBLIC IsEmpty : BOOL
GET
END_GET
END_PROPERTY

{attribute 'monitoring':='call'}
PROPERTY PUBLIC IsFull : BOOL
GET
END_GET
END_PROPERTY

METHOD PUBLIC ResetIterator : BOOL
VAR_INPUT
END_VAR
END_METHOD

//Restore the iterator to the value before the last reset. This is necessary if several white loops are placed inside each other
METHOD PUBLIC RestoreIterator : BOOL
VAR_INPUT
END_VAR
END_METHOD

{attribute 'monitoring':='call'}
PROPERTY PUBLIC Size : UDINT
GET
END_GET
END_PROPERTY

END_INTERFACE
